FUNCTION_BLOCK FB_Add
VAR_IN_OUT
    iValue : INT;
END_VAR


VAR
    normalVar : INT := 0;
END_VAR

VAR_TEMP
    tempVar : INT;
END_VAR

iValue := iValue + 10;



normalVar := normalVar + 1;
tempVar := tempVar + 1;
//staticVar := staticVar + 1;

END_FUNCTION_BLOCK

(* stored: Version 1.1.0.1, ProductVersion 3.1.4024.16
   POU FB_Add: Id {c050360c-48e5-4dfb-9ac6-5ec662c8ac86}, SpecialFunc None *)
